// TIA Portal V17 export
// export: Created 2023-12-22T15:08:09.9852082Z, ExportSetting WithDefaults, DisplayName Totally Integrated Automation Portal, DisplayVersion V17, DisplayName TIA Portal Openness, DisplayVersion V17, DisplayName TIA Portal Version Control Interface, DisplayVersion V17, DisplayName STEP 7 Professional, DisplayVersion V17, DisplayName STEP 7 Safety, DisplayVersion V17, DisplayName WinCC Advanced, DisplayVersion V17
DATA_BLOCK "Logick_DB"   // DB1
VERSION : 0.1
// stored: AutoNumber true, DBAccessibleFromOPCUA true, DBAccessibleFromWebserver true, InstanceOfName Logick, InstanceOfType FB
"Logick"
   // VAR_INPUT
   //    PE : Real;
   //    LE_Target : Real;
   //    LE_Source : Real;
   // END_VAR
   // VAR RETAIN
   //    Start : Bool;
   //    Dynamic : Bool;
   //    Rotation : Bool;
   //    Load : Bool;
   //    Reload : Bool;
   //    Deload : Bool;
   //    PS_Add : Bool;
   //    PS_Sub : Bool;
   //    PE_Alarm : Bool;
   //    PE_Warning : Bool;
   //    LE_in_Alarm : Bool;
   //    LE_in_Warning : Bool;
   //    LE_out_Alarm : Bool;
   //    LE_out_Warning : Bool;
   //    Mode { S7_SetPoint := 'True'} : Int := 1;
   //    "Step" : Int;
   //    SP_Hz : Real;
   //    PS_REQ : Int;
   //    PS_cnt : Int;
   //    PE_SP { S7_SetPoint := 'True'} : Real := 14.5;
   //    PE_StartUp : Real;
   //    PE_Work : Real;
   //    LE_Target_SP : Real;
   //    LE_Source_SP : Real := 3.65;
   //    PID_Correction : Real;
   //    SP_Low : Real;
   //    SP_High { S7_SetPoint := 'True'} : Real := 42.0;
   //    SP_Min { S7_SetPoint := 'True'} : Real := 12.0;
   //    SP_PE_Alarm { S7_SetPoint := 'True'} : Real := 22.0;
   //    SP_PE_Warning { S7_SetPoint := 'True'} : Real := 20.0;
   //    SP_LE_in_Warning { S7_SetPoint := 'True'} : Real := 1.85;
   //    SP_LE_in_Alarm { S7_SetPoint := 'True'} : Real := 1.2;
   //    SP_LE_out_Warning { S7_SetPoint := 'True'} : Real := 1.0;
   //    SP_LE_out_Alarm { S7_SetPoint := 'True'} : Real := 2.0;
   //    xPE : Real;
   //    xPE_Min { S7_SetPoint := 'True'} : Real := 0.7;
   //    Mode_5_REQ { S7_SetPoint := 'True'} : Int := 2;
   //    Mode_5_SP { S7_SetPoint := 'True'} : Real := 44.4;
   //    in_PE_LS { S7_SetPoint := 'True'} : Real := -0.4;
   //    in_PE_LLS { S7_SetPoint := 'True'} : Real := -0.8;
   //    Events : Word;
   //    Alarms : Word;
   //    pos : Array[0..15] of Bool;
   //    T_Delay_ADD { S7_SetPoint := 'True'} : "Time_M";
   //    T_Delay_SUB { S7_SetPoint := 'True'} : "Time_M";
   //    T_Rotation { S7_SetPoint := 'True'} : "Time_D";
   //    T_in_PE { S7_SetPoint := 'True'} : "Time_M";
   // END_VAR
BEGIN
   T_Delay_ADD.SP_M := 5;
   T_Delay_ADD.SP_S := 0;
   T_Delay_SUB.SP_M := 5;
   T_Delay_SUB.SP_S := 0;
   T_Rotation.SP_D := 7;
   T_Rotation.SP_H := 0;
   T_Rotation.SP_M := 2;
   T_Rotation.SP_S := 0;
   T_in_PE.SP_M := 0;
   T_in_PE.SP_S := 30;
END_DATA_BLOCK
